// Mitsubishi GX Works2 project: LRI - PLC - AND   PLC: Q03UDV

PROGRAM MAIN
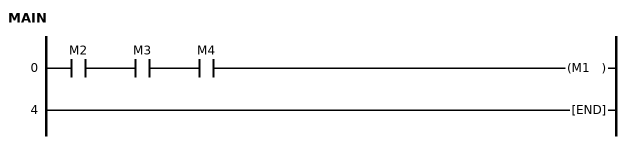
0     LD      M2
      AND     M3
      AND     M4
      OUT     M1
4     END
END_PROGRAM
